// TIA Portal V20 export
FUNCTION_BLOCK "FB_Frequency_Inverter"   // FB6, LAD
{ S7_Optimized_Access := 'TRUE' }
// stored: AutoNumber false, MemoryReserve 100, SetENOAutomatically false
   VAR_INPUT
      Emergency_Stop_Release : Bool;
      Start : Bool;
      Manual_Turn_On_Motor : Bool;
      Pause_Conveyor_Belt_And_Carousel_Functional_Test : Bool;
      Select_Motor_Speedy : SInt;
   END_VAR
   VAR_OUTPUT
      Motor_Spining_Speedy_1 : Bool;
      Motor_Spining_Speedy_2 : Bool;
      Motor_Spining_Speedy_3 : Bool;
   END_VAR
BEGIN

REGION Network 1
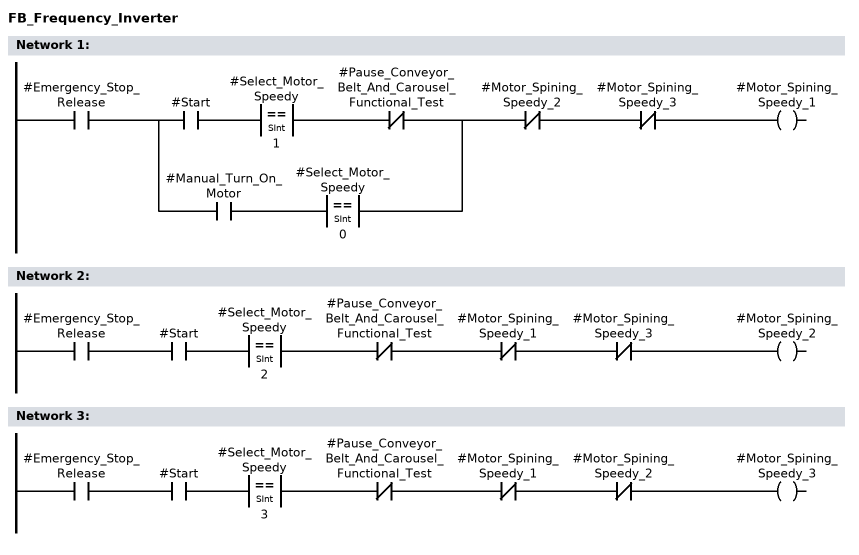
   RUNG wire#powerrail
      Contact( #Emergency_Stop_Release )
      wire#w1
      Contact( #Start )
      { S7_Templates := "SrcType := SInt" } EQ_Contact(in1 := #Select_Motor_Speedy, in2 := 1)
      I_Contact( #Pause_Conveyor_Belt_And_Carousel_Functional_Test )
      wire#w2
      I_Contact( #Motor_Spining_Speedy_2 )
      I_Contact( #Motor_Spining_Speedy_3 )
      Coil( #Motor_Spining_Speedy_1 )
   END_RUNG
   RUNG wire#w1
      Contact( #Manual_Turn_On_Motor )
      { S7_Templates := "SrcType := SInt" } EQ_Contact(in1 := #Select_Motor_Speedy, in2 := 0)
   END_RUNG wire#w2
   // the same network as SCL:
   #Motor_Spining_Speedy_1 := #Emergency_Stop_Release AND ((#Start AND (#Select_Motor_Speedy = 1) AND NOT #Pause_Conveyor_Belt_And_Carousel_Functional_Test) OR (#Manual_Turn_On_Motor AND (#Select_Motor_Speedy = 0))) AND NOT #Motor_Spining_Speedy_2 AND NOT #Motor_Spining_Speedy_3;
END_REGION

REGION Network 2
   RUNG wire#powerrail
      Contact( #Emergency_Stop_Release )
      Contact( #Start )
      { S7_Templates := "SrcType := SInt" } EQ_Contact(in1 := #Select_Motor_Speedy, in2 := 2)
      I_Contact( #Pause_Conveyor_Belt_And_Carousel_Functional_Test )
      I_Contact( #Motor_Spining_Speedy_1 )
      I_Contact( #Motor_Spining_Speedy_3 )
      Coil( #Motor_Spining_Speedy_2 )
   END_RUNG
   // the same network as SCL:
   #Motor_Spining_Speedy_2 := #Emergency_Stop_Release AND #Start AND (#Select_Motor_Speedy = 2) AND NOT #Pause_Conveyor_Belt_And_Carousel_Functional_Test AND NOT #Motor_Spining_Speedy_1 AND NOT #Motor_Spining_Speedy_3;
END_REGION

REGION Network 3
   RUNG wire#powerrail
      Contact( #Emergency_Stop_Release )
      Contact( #Start )
      { S7_Templates := "SrcType := SInt" } EQ_Contact(in1 := #Select_Motor_Speedy, in2 := 3)
      I_Contact( #Pause_Conveyor_Belt_And_Carousel_Functional_Test )
      I_Contact( #Motor_Spining_Speedy_1 )
      I_Contact( #Motor_Spining_Speedy_2 )
      Coil( #Motor_Spining_Speedy_3 )
   END_RUNG
   // the same network as SCL:
   #Motor_Spining_Speedy_3 := #Emergency_Stop_Release AND #Start AND (#Select_Motor_Speedy = 3) AND NOT #Pause_Conveyor_Belt_And_Carousel_Functional_Test AND NOT #Motor_Spining_Speedy_1 AND NOT #Motor_Spining_Speedy_2;
END_REGION
END_FUNCTION_BLOCK
